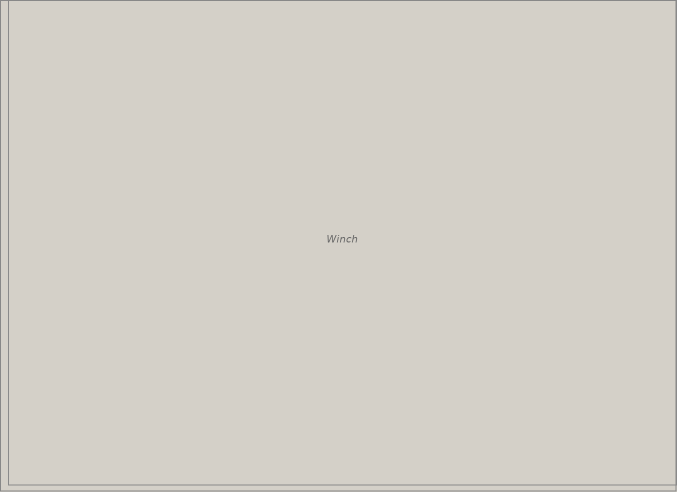
VISUALIZATION Main  // 677x492
    TabControl (8,-7 669x492)
        shows Winch()
        shows Cylinder()
        [0]: TabTitle=Winch
        [1]: TabTitle=Cylinder
END_VISUALIZATION

(* stored: Version 1.1.0.1, ProductVersion 3.1.4024.11
   Visu Main: Id {c8398d6f-4ceb-4850-a46d-48fbc6c4726c} *)
